PROGRAM MACHINE
VAR
END_VAR



IF bMAIN_RESET THEN
	iMAIN_STATE:=98 ;
	bMAIN_PAUSE:=FALSE;
END_IF

END_PROGRAM

(* stored: Version 1.1.0.1, ProductVersion 3.1.4024.12
   POU MACHINE: Id {9f31af90-0ebb-4c9c-9f88-fd85631a41cf}, SpecialFunc None *)
